// TwinCAT 3 PLC project Aufgabe3
// ProgramVersion: 3.1.4023.0
// libraries:
//   Tc2_Standard, * (Beckhoff Automation GmbH)
//   Tc2_System, * (Beckhoff Automation GmbH)
//   Tc3_Module, * (Beckhoff Automation GmbH)
// project tree:
//   GVLs/ GVL_IO.TcGVL
//   / PlcTask.TcTTO
//   POUs/ MAIN.TcPOU
// (motion and I/O tree: see PLC project aufgabe1)
// real-time tasks:
//   TASK PlcTask: cycle T#1ms, priority 1, ADS port 350
//   TASK FastTask: cycle T#300us, priority 2, ADS port 351
//   TASK SlowTask: cycle T#10ms, priority 3, ADS port 352
//   TASK PlcTask1: cycle T#10ms, priority 20, ADS port 353
// variable links:
//   Aufgabe3/Aufgabe3 Instance <-> Device 1 (EtherCAT)/Term 1 (EK1100)/Term 2 (EL2004)
//     PlcTask Outputs/GVL_IO.DO_LampGreen <-> Channel 2/Output
//     PlcTask Outputs/GVL_IO.DO_LampOrange <-> Channel 3/Output
//     PlcTask Outputs/GVL_IO.DO_LampRed <-> Channel 1/Output
//   Aufgabe3/Aufgabe3 Instance <-> Device 1 (EtherCAT)/Term 1 (EK1100)/Term 3 (EL1004)
//     PlcTask Inputs/GVL_IO.DI_BtnBlue <-> Channel 2/Input
//     PlcTask Inputs/GVL_IO.DI_BtnGreen <-> Channel 3/Input
//     PlcTask Inputs/GVL_IO.DI_BtnYellow <-> Channel 1/Input

CONFIGURATION Aufgabe3
    RESOURCE PLC ON TwinCAT3
        TASK PlcTask(INTERVAL := T#10ms, PRIORITY := 20);
        PROGRAM MAIN WITH PlcTask : MAIN;
    END_RESOURCE
END_CONFIGURATION

// ---- GVLs/GVL_IO.TcGVL
{attribute 'qualified_only'}
VAR_GLOBAL
	DI_BtnYellow    AT %I* : BOOL;
    DI_BtnBlue      AT %I* : BOOL;
	DI_BtnGreen     AT %I* : BOOL;
    
    DO_LampRed      AT %Q* : BOOL;
    DO_LampGreen    AT %Q* : BOOL;
	DO_LampOrange   AT %Q* : BOOL;
END_VAR

// ---- POUs/MAIN.TcPOU
PROGRAM MAIN
VAR
END_VAR

END_PROGRAM
